Fanuc KAREL source: kt00152.KL

-- PROVISIONAL review KL for V940-1; original PC SHA256 46284f78ce56ba2e785c94a3811e09cc0c3d3e73baf18b3dab0e6df64a20afdb
-- Incomplete behavior may be omitted. Consult companion uncertainty JSON. Do not deploy.
PROGRAM KT00152
%NOLOCKGROUP
VAR
  OUT : REAL
-- UNRESOLVED_DECL Y1 type=002018
-- UNRESOLVED_DECL H2 type=002017
BEGIN
  -- V9_ZERO_TABLE_METADATA_HINT layout=0001; no indexed target words; source/name/runtime held
  -- UNRESOLVED_PC offsets 5-19; opcodes 2E,22,9D,33,B2
  -- UNRESOLVED_PC offsets 24-38; opcodes 2E,22,9D,33,B4
  -- UNRESOLVED_PC offsets 43-69; opcodes 22,9D,33,B1,22,9D,33,B3,55,64,23
  -- UNRESOLVED_PC offsets 74-78; opcodes 7F
END KT00152
